// TIA Portal V20 export
TYPE "LBP_typeHMI"
TITLE = Operator panel signals / Signaux pupitre opérateur
// User data type for block LBP_HMI [DB19] / Type de données utilisateur pour bloc LBP_HMI [DB19]
   STRUCT
      A_SCLight : Bool;   // Screen light / Éclaircir écran
      A_SCDark : Bool;   // Screen darkening / Obscurcissement écran
      A_KeyDisable : Bool;   // Key disable / Désactiver touche
      A_ClearCanAl : Bool;   // Clear cancel alarms / Supprimer alarmes d'abandon
      A_ClearRecAl : Bool;   // Clear recall alarms / Supprimer alarmes de rappel
      f0_5 : Bool;
      A_SafeActionLog : Bool;   // Edge change 0 → 1: Save ACTION.COM to CRASH.COM / Front 0 → 1 : enregistrer ACTION.COM dans CRASH.COM
      A_ActWCS : Bool;   // Actual value in WCS 0=MCS / Valeur réelle dans WCS 0=MCS
      A_PLCExtViewerReject : Bool;   // External viewer reject / Refuser visualiseur externe
      A_PLCExtViewerMode : Bool;   // External viewer mode / Mode visualiseur externe
      f1_2 : Bool;
      f1_3 : Bool;
      f1_4 : Bool;
      f1_5 : Bool;
      f1_6 : Bool;
      f1_7 : Bool;
      A_1stError1 : Word;   // 1st error HIGRAPH / 1re erreur HIGRAPH
      A_1stError2 : Word;   // 1st error HIGRAPH / 1re erreur HIGRAPH
      A_ASpi1percent : Byte;   // Analog spindle 1: / Broche analogique 1 :
      A_ASpi2percent : Byte;
      A_MCPChan : Byte;
      A_OEM1 : Bool;
      A_OEM2 : Bool;
      A_AToolMeas : Bool;   // AutoToolMeasure
      f9_3 : Bool;
      f9_4 : Bool;
      f9_5 : Bool;
      f9_6 : Bool;
      f9_7 : Bool;
      A_Hardkey : Byte;   // PLC hardkeys / Touches matérielles AP
      f11 : Byte;   // Reserved for hardkeys / Réservé pour touches matérielles
      f12_0 : Bool;
      f12_1 : Bool;
      A_COM2 : Bool;
      A_COM1 : Bool;
      A_V24stop : Bool;
      A_V24ext : Bool;
      A_V24off : Bool;
      A_V24on : Bool;
      A_TeachDisable : Bool;
      f13_1 : Bool;
      f13_2 : Bool;
      f13_3 : Bool;
      f13_4 : Bool;
      A_PPdeload : Bool;
      A_PPload : Bool;
      A_PPsel : Bool;
      A_V24Index1 : Byte;
      A_V24Index2 : Byte;
      A_V24NoFile1 : Byte;
      A_V24NoFile2 : Byte;
      A_res18 : Byte;
      A_res19 : Byte;   // Message counter / Compteur de messages
      f20_0 : Bool;
      E_SCDark : Bool;   // Screen darkening / Obscurcissement écran
      E_Cancel : Bool;   // Cancel / Abandon
      E_CanCleared : Bool;   // Cancel alarms cleared / Alarmes d'abandon supprimées
      E_RecCleared : Bool;   // Recall alarms cleared / Alarmes de rappel supprimées
      f20_5 : Bool;   // res. language / rés. langue
      E_SimActiv : Bool;   // Simulation active
      E_ActWCS : Bool;   // Switchover MCS/WCS 0=MCS / Commutation MCS/WCS 0=MCS
      E_ActivWA : Byte;
      E_Chan : Byte;   // Channel displayed / Canal affiché
      E_KeybHandl : Bool;   // Keyboard handling / Gestion clavier
      E_DataTransf : Bool;   // Data transfer active / Transmission de données active
      E_DisplChange : Bool;   // Display change / Modification affichage
      f23_3 : Bool;
      f23_4 : Bool;
      f23_5 : Bool;
      f23_6 : Bool;
      f23_7 : Bool;
      E_ScreenNo : Word;
      E_res26_0 : Bool;   // Reserved / Réservé
      E_PPOK : Bool;   // Part program status OK / État programme pièce OK
      E_PPErr : Bool;   // Part program status error / Programme pièce erreur d'état
      E_PPAct : Bool;   // Part program status active / État programme pièce actif
      f26_4 : Bool;   // Reserved / Réservé
      E_PPdeload : Bool;   // Part program status deloading / État programme pièce en cours de déchargement
      E_PPload : Bool;   // Part program status loading / État programme pièce en cours de chargement
      E_PPsel : Bool;   // Part program status selecting / État programme pièce en cours de sélection
      E_PPError : Byte;   // Part program status error / Programme pièce erreur d'état
      A_PictNo : Int;
      A_PictOn : Bool;
      A_PictOff : Bool;
      f30_2 : Bool;
      f30_3 : Bool;
      f30_4 : Bool;
      f30_5 : Bool;
      f30_6 : Bool;
      f30_7 : Bool;
      E_PictOK : Bool;
      E_PictOn : Bool;
      E_PictAct : Bool;
      E_PictOff : Bool;
      E_PictErr : Bool;
      f31_5 : Bool;
      f31_6 : Bool;
      E_NotAct : Bool;
      A_FuncNo : Byte;
      A_Par1 : Byte;
      A_Par2 : Byte;
      A_Par3 : Byte;
      E_FuncErr : Byte;
      f37 : Byte;
      f38 : Byte;
      f39 : Byte;
      res40 : Array[0..9] of Byte;
      MMC2 : Struct
         A_SCLight : Bool;   // Screen light / Éclaircir écran
         A_SCDark : Bool;   // Screen darkening / Obscurcissement écran
         A_KeyDisable : Bool;   // Key disable / Désactiver touche
         A_ClearCanAl : Bool;   // Clear cancel alarms / Supprimer alarmes d'abandon
         A_ClearRecAl : Bool;   // Clear recall alarms / Supprimer alarmes de rappel
         f0_5 : Bool;
         f0_6 : Bool;
         A_ActWCS : Bool;   // Actual value in WCS 0=MCS / Valeur réelle dans WCS 0=MCS
         A_PLCExtViewerReject : Bool;   // External viewer reject / Refuser visualiseur externe
         A_PLCExtViewerMode : Bool;   // External viewer mode / Mode visualiseur externe
         f1_2 : Bool;
         f1_3 : Bool;
         f1_4 : Bool;
         f1_5 : Bool;
         f1_6 : Bool;
         f1_7 : Bool;
         A_1stError1 : Word;   // 1st error HIGRAPH / 1re erreur HIGRAPH
         A_1stError2 : Word;   // 1st error HIGRAPH / 1re erreur HIGRAPH
         A_ASpi1percent : Byte;   // Analog spindle 1: / Broche analogique 1 :
         A_ASpi2percent : Byte;
         A_MCPChan : Byte;
         A_OEM1 : Bool;
         A_OEM2 : Bool;
         A_AToolMeas : Bool;   // AutoToolMeasure
         f9_3 : Bool;
         f9_4 : Bool;
         f9_5 : Bool;
         f9_6 : Bool;
         f9_7 : Bool;
         A_Hardkey : Byte;   // PLC hardkeys / Touches matérielles AP
         f11 : Byte;   // Reserved for hardkeys / Réservé pour touches matérielles
         f12_0 : Bool;
         f12_1 : Bool;
         A_COM2 : Bool;
         A_COM1 : Bool;
         A_V24stop : Bool;
         A_V24ext : Bool;
         A_V24off : Bool;
         A_V24on : Bool;
         A_TeachDisable : Bool;
         f13_1 : Bool;
         f13_2 : Bool;
         f13_3 : Bool;
         f13_4 : Bool;
         A_PPdeload : Bool;
         A_PPload : Bool;
         A_PPsel : Bool;
         A_V24Index1 : Byte;
         A_V24Index2 : Byte;
         A_V24NoFile1 : Byte;
         A_V24NoFile2 : Byte;
         A_res18 : Byte;
         A_res19 : Byte;   // Message counter / Compteur de messages
         f20_0 : Bool;
         E_SCDark : Bool;   // Screen darkening / Obscurcissement écran
         E_Cancel : Bool;   // Cancel / Abandon
         E_CanCleared : Bool;   // Cancel alarms cleared / Alarmes d'abandon supprimées
         E_RecCleared : Bool;   // Recall alarms cleared / Alarmes de rappel supprimées
         f20_5 : Bool;   // res. language / rés. langue
         E_SimActiv : Bool;   // Simulation active
         E_ActWCS : Bool;   // Switchover MCS/WCS 0=MCS / Commutation MCS/WCS 0=MCS
         E_ActivWA : Byte;
         E_Chan : Byte;   // Channel displayed / Canal affiché
         E_KeybHandl : Bool;   // Keyboard handling / Gestion clavier
         E_DataTransf : Bool;   // Data transfer active / Transmission de données active
         E_DisplChange : Bool;   // Display change / Modification affichage
         f23_3 : Bool;
         f23_4 : Bool;
         f23_5 : Bool;
         f23_6 : Bool;
         f23_7 : Bool;
         E_ScreenNo : Word;
         E_res26_0 : Bool;   // Reserved / Réservé
         E_PPOK : Bool;   // Part program status OK / État programme pièce OK
         E_PPErr : Bool;   // Part program status error / Programme pièce erreur d'état
         E_PPAct : Bool;   // Part program status active / État programme pièce actif
         f26_4 : Bool;   // Reserved / Réservé
         E_PPdeload : Bool;   // Part program status deloading / État programme pièce en cours de déchargement
         E_PPload : Bool;   // Part program status loading / État programme pièce en cours de chargement
         E_PPsel : Bool;   // Part program status selecting / État programme pièce en cours de sélection
         E_PPError : Byte;   // Part program status error / Programme pièce erreur d'état
         A_PictNo : Int;
         A_PictOn : Bool;
         A_PictOff : Bool;
         f30_2 : Bool;
         f30_3 : Bool;
         f30_4 : Bool;
         f30_5 : Bool;
         f30_6 : Bool;
         f30_7 : Bool;
         E_PictOK : Bool;
         E_PictOn : Bool;
         E_PictAct : Bool;
         E_PictOff : Bool;
         E_PictErr : Bool;
         f31_5 : Bool;
         f31_6 : Bool;
         E_NotAct : Bool;
         A_FuncNo : Byte;
         A_Par1 : Byte;
         A_Par2 : Byte;
         A_Par3 : Byte;
         E_FuncErr : Byte;
         f37 : Byte;
         f38 : Byte;
         f39 : Byte;
         res40 : Array[0..9] of Byte;
      END_STRUCT;
      ONL_REQUEST : Word;
      ONL_CONFIRM : Word;
      PAR_CLIENT_IDENT : Word;
      PAR_MMC_TYP : Byte;
      PAR_MSTT_ADR : Byte;
      PAR_STATUS : Byte;
      PAR_Z_INFO : Byte;
      MtoNAlive : Word;
      f112 : Byte;
      ParOpKeyAdr : Byte;
      ParTcuIndex : Byte;
      f115 : Byte;
      Tcu1KeyAdr : Byte;
      Tcu2KeyAdr : Byte;
      Tcu1Index : Byte;
      Tcu2Index : Byte;
      MMC1_CLIENT_IDENT : Word;
      MMC1_TYP : Byte;
      MMC1_MSTT_ADR : Byte;
      MMC1_STATUS : Byte;
      MMC1_Z_INFO : Byte;
      MMC1_SHIFT_LOCK : Bool;
      MMC1_MSTT_SHIFT_LOCK : Bool;
      MMC1_ACTIVE_REQ : Bool;
      MMC1_ACTIVE_PERM : Bool;
      MMC1_ACTIVE_CHANGED : Bool;
      MMC1_CHANGED_DENIED : Bool;
      MMC1_TCU_SHIFT_LOCK : Bool;
      f127 : Byte;
      MMC1_TRANS_DB : Word;
      MMC2_CLIENT_IDENT : Word;
      MMC2_TYP : Byte;
      MMC2_MSTT_ADR : Byte;
      MMC2_STATUS : Byte;
      MMC2_Z_INFO : Byte;
      MMC2_SHIFT_LOCK : Bool;
      MMC2_MSTT_SHIFT_LOCK : Bool;
      MMC2_ACTIVE_REQ : Bool;
      MMC2_ACTIVE_PERM : Bool;
      MMC2_ACTIVE_CHANGED : Bool;
      MMC2_CHANGED_DENIED : Bool;
      MMC2_TCU_SHIFT_LOCK : Bool;
      f137 : Byte;
      MMC2_TRANS_DB : Word;
      A_Subtype : Int;   // For code carrier Input from PLC / Pour porte-code entrée par AP
      A_Duplo : Int;
      A_Ident : String[32];
      A_Tnumber : Int;
      A_MagazinePlace : Int;
      A_MagazinePlaceType : Int;
      A_ToolSize_Upper : Byte;
      A_ToolSize_Down : Byte;
      A_ToolSize_Left : Byte;
      A_ToolSize_Right : Byte;
      A_Channel : Byte;
      A_LoadingPlace : Byte;
      A_Magazine : Int;
      A_Unit : Byte;
      A_NCU_Index : Byte;
      A_FileIndex : Int;
      A_ActiveEnable : Bool;
      A_Override : Bool;
      A_LoadTool : Bool;
      A_DeleteTool : Bool;
      E_Subtype : Int;   // For code carrier Output to PLC / Pour porte-code sortie vers AP
      E_Duplo : Int;
      E_Ident : String[32];
      E_Tnumber : Int;
      E_ToolState : Int;
      E_MagazinePlaceType : Int;
      E_ToolSize_Upper : Byte;
      E_ToolSize_Down : Byte;
      E_ToolSize_Left : Byte;
      E_ToolSize_Right : Byte;
      E_Magazine : Int;
      E_MagazinePlace : Int;
      A_ReqMMC1 : Bool;   // For code carrier Request MMC-Interface1 / Pour porte-code demander interface MMC1
      A_ReqMMC2 : Bool;   // For code carrier Request MMC-Interface2 / Pour porte-code demander interface MMC2
      A_K_Code : Byte;
      E_Done : Bool;
      E_Error : Bool;
      E_Active : Bool;
      f252_3 : Bool;
      f252_4 : Bool;
      f252_5 : Bool;
      f252_6 : Bool;
      E_Ident_Ready : Bool;
      E_K_CodeError : Byte;   // Identify for Error_Code / Identifier pour Error_Code
      E_Error_Code : Int;
      E_Req : Bool;   // For Positioning / Pour positionnement
      f257 : Byte;
      A_Done : Bool;
      A_Error : Bool;
      A_Active : Bool;
      f258_3 : Bool;
      f258_4 : Bool;
      f258_5 : Bool;
      f258_6 : Bool;
      f258_7 : Bool;
      E_TDC_Read : Bool;
      E_TDC_Write : Bool;
      E_TDC_Cancel : Bool;
      E_TDC_Read_before_Write : Bool;
      f259_4 : Bool;
      f259_5 : Bool;
      f259_6 : Bool;
      f259_7 : Bool;
      A_Error_Code : Int;
      E_PMagazine : Int;
      E_PMagazinePlace : Int;
      E_PTnumber : Int;   // TPM data / Données TPM
      A_TPMStatus : Int;
      A_TPMCounter : Array[1..32] of DInt;
      A_HWeelSimOvr : Byte;
      f399 : Byte;
      A_SimOvr : Int;   // Simulation override / Correction simulation
      A_SimState : Int;   // Simulation state / État simulation
      E_HmiUserKey : Array[1..64] of Bool;   // HMI user keys for HMI sidescreen / HMI touches utilisateur pour écran latéral IHM
      A_HmiUserLed : Array[1..64] of Bool;   // LEDs to the user keys for HMI sidescreen / LED pour touches utilisateur pour écran latéral IHM
      A_DisableHmiUserKey : Array[1..64] of Bool;   // Disable user keys for HMI sidescreen / Désactiver les touches utilisateur pour écran latéral IHM
      SafetyAutoAcceptanceTest : Struct   // Interface for the automated acceptance test
         E_Prepare : Bool;   // Prepare automated acceptance test requested by client
         E_Finalize : Bool;   // Stop automated acceptance test requested by client
         E_Cancel : Bool;   // Cancel automated acceptance test requested by client
         E_Perform : Bool;   // Perform automated acceptance test requested by client
         E_PerformSequence : Bool;   // Perform entire test sequence for automated acceptance test requested by client
         f428_5 : Bool;
         f428_6 : Bool;
         f428_7 : Bool;
         f429 : Byte;
         A_Prepared : Bool;   // Automated acceptance test was successfully prepared
         A_Finalized : Bool;   // Automated acceptance test was successfully stopped
         A_Canceled : Bool;   // Automated acceptance test was canceled successfully
         A_Performed : Bool;   // Automated acceptance test was performed successfully
         A_SequencePerformed : Bool;   // Entire test sequence for automated acceptance test is running
         f430_5 : Bool;
         f430_6 : Bool;
         f430_7 : Bool;
         f431_0 : Bool;
         A_Error : Bool;   // Automated acceptance test was canceled
         A_InvalidGroup : Bool;   // Test group is not accepted
         A_InvalidNumber : Bool;   // Test number is not accepted
         f431_4 : Bool;
         f431_5 : Bool;
         f431_6 : Bool;
         f431_7 : Bool;
         E_Group : Int;   // Test group for the current test
         E_Number : Int;   // Test number for the current test
         E_AxisNumber : Int;   // Axis number for the current test
         E_TraversePlus : Bool;   // Traversing direction for the current test (FALSE=negative, TRUE=positive)
         E_SelectSafeStop : Bool;   // Safe Stop is set for the current test
         E_SelectBrake : Bool;   // Brake used for the current test. (FALSE=Brake1, TRUE=Brake2)
         E_SelectSbtMode : Bool;   // SBT Test Sequence used for the current test. (FALSE=Sequence1, TRUE=Sequence2)
         E_SelectSlpMode : Int;   // Safe End Position used for the current test. ("SE/SLP PositionArea" : 1=SE1 ; 2=SE2)
         E_SelectSlsMode : Int;   // Safe Speed (SG1..SG4) used for the current test
      END_STRUCT;
   END_STRUCT;
END_TYPE
